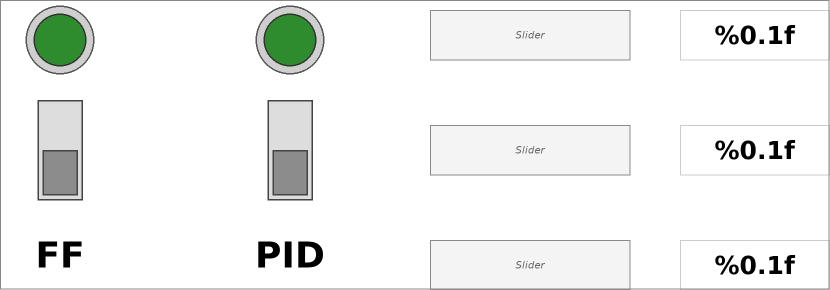
VISUALIZATION VISU_ControlFeatures  // 830x290
    DipSwitch (240,100 100x100), variable: bValve, behaviour: TOGGLE, style: Switch-DipSwitch-Gray
    Lamp1 (250,0 80x80), variable: bValveLamp, style: Lamp-Lamp1-Green
    Textfield (230,230 120x50), "PID"
    DipSwitch (10,100 100x100), variable: bFeedForward, behaviour: TOGGLE, style: Switch-DipSwitch-Gray
    Lamp1 (20,0 80x80), variable: bFFLamp, style: Lamp-Lamp1-Green
    Textfield (0,230 120x50), "FF"
    Slider (430,125 200x50), variable: fSliderKi, scale 0..10
    Slider (430,240 200x50), variable: fSliderKd, scale 0..5
    Textfield (680,10 150x50), "%0.1f", text variable: G_Parameter.Kp
    Textfield (680,125 150x50), "%0.1f", text variable: G_Parameter.Ki
    Textfield (680,240 150x50), "%0.1f", text variable: G_Parameter.Kd
    Slider (430,10 200x50), variable: fSliderKp, scale 0..30
END_VISUALIZATION

(* stored: Version 1.1.0.1
   Visu VISU_ControlFeatures: Id {98b30c8c-8faa-4088-b126-74a040433228} *)
